PROGRAM Tsk_MAIN_10ms
VAR

END_VAR

END_PROGRAM

(* stored: Version 1.1.0.1, ProductVersion 3.1.4024.11
   POU Tsk_MAIN_10ms: Id {0c28050e-c50b-4e4d-8e0a-6abe193c6a93}, SpecialFunc None *)
